FUNCTION_BLOCK FB_TelescopeState IMPLEMENTS I_TelescopeState
VAR_INPUT
END_VAR
VAR_OUTPUT
END_VAR
VAR
	pMachine 		: POINTER TO FB_TelescopeMachine;
	comm			: I_Comm;
	
	bInitialize		: BOOL;
	bPark			: BOOL;
	bReset			: BOOL;
	bSlew			: BOOL;
	bStop			: BOOL;
	bTrack			: BOOL;
	iStage			: UINT;
END_VAR

METHOD FB_init : BOOL
VAR_INPUT
	bInitRetains 	: BOOL; // if TRUE, the retain variables are initialized (warm start / cold start)
	bInCopyCode 	: BOOL;  // if TRUE, the instance afterwards gets moved into the copy code (online change)
	pMachine 		: POINTER TO FB_TelescopeMachine;
	comm			: I_Comm;	
END_VAR
THIS^.pMachine := pMachine;
THIS^.comm := comm;
END_METHOD

METHOD Initialize : BOOL
VAR_INPUT
END_VAR
bInitialize := TRUE;
END_METHOD

METHOD Park : BOOL
VAR_INPUT
END_VAR
bPark := TRUE;
iStage := 0;
END_METHOD

METHOD Reset : BOOL
VAR_INPUT
END_VAR
bReset := TRUE;
iStage := 0;
END_METHOD

METHOD Slew : BOOL
VAR_INPUT
	fAzimuth	: LREAL;
	fAltitude	: LREAL;
END_VAR
bSlew := TRUE;
iStage := 0;
END_METHOD

METHOD Stop : BOOL
VAR_INPUT
END_VAR
bStop := TRUE;
iStage := 0;
END_METHOD

METHOD Track : BOOL
VAR_INPUT
	fRightAscension	: LREAL;
	fDeclination	: LREAL;
END_VAR
bTrack := TRUE;
iStage := 0;
END_METHOD

END_FUNCTION_BLOCK

(* stored: Version 1.1.0.1, ProductVersion 3.1.4024.15
   POU FB_TelescopeState: Id {a1655b2a-b366-4c97-b1c5-df3d2b5e068d}, SpecialFunc None
   Method FB_init: Id {939ce836-b748-4327-8af4-fef7b1a3e467}
   Method Initialize: Id {4014e65c-f049-46d7-ab38-f9d8532488b1}
   Method Park: Id {1d7b2094-1b9e-4f3f-8684-35da700e0b9a}
   Method Reset: Id {57d7d305-bed4-400e-bbf9-c181dc7d793e}
   Method Slew: Id {e5dd4f78-c7c2-4163-9dee-c9e4a43c707b}
   Method Stop: Id {f88b6084-031f-4751-912f-ee2fd3d7f783}
   Method Track: Id {33662814-9536-4e5d-81b1-cbf07479cb1d} *)
